INTERFACE I_SpscBuffer

PROPERTY Capacity : UDINT
GET
END_GET
END_PROPERTY

METHOD Clear
VAR_INPUT
END_VAR
END_METHOD

PROPERTY Empty : bool
GET
END_GET
END_PROPERTY

PROPERTY Full : bool
GET
END_GET
END_PROPERTY

METHOD Get : BOOL
VAR_INPUT
	pDestination 	: pvoid;
	cbSize 			: UDINT;
END_VAR
END_METHOD

METHOD Initialize : BOOL
VAR_INPUT
	nElementSize 		: UDINT;
	nElementCapacity 	: UDINT;
END_VAR
END_METHOD

METHOD Push : BOOL
VAR_INPUT
	pData : pvoid;
	cbSize : UDINT;
END_VAR
END_METHOD

METHOD Reset
END_METHOD

PROPERTY Size : UDINT
GET
END_GET
END_PROPERTY

END_INTERFACE

(* stored: Version 1.1.0.1
   Itf I_SpscBuffer: Id {c99df50e-d85d-49db-9b2a-956615e26b28}
   Property Capacity: Id {74e5f4fb-c854-4aec-8dfd-467fbf66a0a3}
   Get Get: Id {9b99bc61-6150-4aa6-bb76-0d9fea28faea}
   Method Clear: Id {5ca14bc2-2bce-48a1-b9b9-b3f5b94ee5b4}
   Property Empty: Id {ec2ff1ec-537c-42d2-9ffc-80c6ca8b5245}
   Get Get: Id {8726a545-4f29-440e-b355-e0669d318b0f}
   Property Full: Id {a9897bab-0747-4d6c-b4a5-473b00e24744}
   Get Get: Id {c592efff-c880-4960-a443-f6b550b3ae72}
   Method Get: Id {25bb8191-df61-414c-b6bf-731edf9f5b48}
   Method Initialize: Id {f6f1f3a0-27ca-4d2d-88dd-ff200ca83243}
   Method Push: Id {9efd7012-eac9-4a55-a179-b16e052d1641}
   Method Reset: Id {75844e62-151e-410e-bfde-488e8008a937}
   Property Size: Id {f37009f0-0d21-4024-8039-9c5989d2a17f}
   Get Get: Id {92bda758-e972-4f11-b02d-4b85e05e3e9e} *)
